// TwinCAT 3 PLC project automatedAquariumfilter
// ProgramVersion: 3.1.4024.0
// libraries:
//   Tc2_Standard, * (Beckhoff Automation GmbH)
//   Tc2_System, * (Beckhoff Automation GmbH)
//   Tc3_Module, * (Beckhoff Automation GmbH)
//   VisuDialogs, * (System)
//   VisuSymbols,3.5.10.0,System
// project tree:
//   FUNCTIONSBLOCKS/ FB_CO2.TcPOU, FB_FILTER.TcPOU, FB_HEATING.TcPOU, FB_LIGHT.TcPOU, FB_WATERCOOLING.TcPOU
//   / GlobalTextList.TcGTLO, GVL.TcGVL, PlcTask.TcTTO, Task_heat.TcTTO, Task_temp_monitor.TcTTO, Visualization Manager.TcVMO (not stored)
//   POUs/ HEATING.TcPOU, MAIN.TcPOU, TEMP_MONITOR.TcPOU
//   VISUs/ Visualization.TcVIS
// real-time tasks:
//   TASK PlcTask: cycle T#10ms, priority 20, ADS port 350

CONFIGURATION automatedAquariumfilter
    RESOURCE PLC ON TwinCAT3
        TASK PlcTask(INTERVAL := T#10ms, PRIORITY := 1);
        TASK Task_heat(INTERVAL := T#10ms, PRIORITY := 3);
        TASK Task_temp_monitor(INTERVAL := T#10ms, PRIORITY := 2);
        PROGRAM MAIN WITH PlcTask : MAIN;
        PROGRAM HEATING WITH Task_heat : HEATING;
        PROGRAM TEMP_MONITOR WITH Task_temp_monitor : TEMP_MONITOR;
    END_RESOURCE
END_CONFIGURATION

// ---- GVL.TcGVL
{attribute 'qualified_only'}
VAR_GLOBAL
	ix_START :BOOL;
	
	ox_FILTER_WATER: BOOL;
	ox_HEATER: BOOL;
	id_TEMP_SENSOR: DINT:=20;
	ix_COOLDOWN: BOOL;
	ix_TEMPRESET: BOOL;
	
	ox_CO2: BOOL;
	ox_LIGHT: BOOL;
	id_TEMP_SETPOINT: DINT:=28;
END_VAR

// ---- POUs/MAIN.TcPOU
PROGRAM MAIN
VAR
	FilterCycle1 : FB_FILTER;  // instantie van FB

	CO2_1:FB_CO2;
	LIGHT1:FB_LIGHT;
	
	
END_VAR

GVL.id_TEMP_SETPOINT:=28;

IF GVL.ix_TEMPRESET THEN
	GVL.id_TEMP_SENSOR := 30;
	GVL.ix_TEMPRESET:=FALSE;
END_IF

IF GVL.ix_COOLDOWN THEN
	GVL.id_TEMP_SENSOR := GVL.id_TEMP_SENSOR -5;
	GVL.ix_COOLDOWN:=FALSE;
END_IF	

GVL.ox_CO2 :=CO2_1.CO2;
GVL.ox_FILTER_WATER := FilterCycle1.FILTER_WATER;
GVL.ox_LIGHT :=LIGHT1.LIGHT;

//FUNCTIEBLOKKEN

FilterCycle1(ix_START := GVL.ix_START);
CO2_1(ix_START :=GVL.ix_START);
LIGHT1(ix_START :=GVL.ix_START);

END_PROGRAM

// ---- FUNCTIONSBLOCKS/FB_FILTER.TcPOU
FUNCTION_BLOCK FB_FILTER
VAR_INPUT
    ix_START : BOOL;  // HMI start input

END_VAR
VAR_OUTPUT
    FILTER_WATER : BOOL;  // output naar MAIN/HMI
END_VAR
VAR
    STATE_FILTER : INT := 0;  // interne state
    T_CYCLE : TON; 
    elapsed_ms : UDINT;  // elapsed time in ms
    cycle_ms   : UDINT;  // 5-second repeating cycle
END_VAR

// --- CASE state machine ---
CASE STATE_FILTER OF

    0: // Idle
        FILTER_WATER := FALSE;

        // Stop cycle timer
        T_CYCLE(IN := FALSE);

        // Start cycle
        IF ix_START THEN
            STATE_FILTER := 1;
        END_IF;

    1: // 30s cycle running
        // Abort cycle if button released
        IF ix_START = FALSE THEN
            STATE_FILTER := 0;
        END_IF;

        // Start 30-second timer
        T_CYCLE(IN := TRUE, PT := T#30S);
	
		// Convert elapsed time to milliseconds
		elapsed_ms := TO_UDINT(T_CYCLE.ET);

		// Create repeating 5-second cycle
		cycle_ms := elapsed_ms MOD 5000; // 5000 ms = 5 seconds
		
		// 0-3s -> ON, 3-5s -> OFF
		IF cycle_ms < 3000 THEN
			FILTER_WATER := TRUE;
		ELSE
			FILTER_WATER := FALSE;
		END_IF;
		        // End of cycle
        IF T_CYCLE.Q THEN
            STATE_FILTER := 0;
        END_IF;
       
END_CASE;

END_FUNCTION_BLOCK

// ---- FUNCTIONSBLOCKS/FB_CO2.TcPOU
FUNCTION_BLOCK FB_CO2
VAR_INPUT
	ix_START: BOOL;
END_VAR
VAR_OUTPUT
	CO2: BOOL;
END_VAR
VAR
	STATE: INT;
	T_CYCLE: TON;
END_VAR

// --- CASE state machine ---
CASE STATE OF

    0: // Idle
        CO2 := FALSE;
        // Stop cycle timer
        T_CYCLE(IN := FALSE);
        // Start cycle
        IF ix_START THEN
            STATE := 1;
        END_IF;
    1: // Start 30s cycle
        // Stop cycle if start button released
        IF ix_START = FALSE THEN
            STATE := 0;
        END_IF;
        // Start timer
        T_CYCLE(IN := TRUE, PT := T#30S);
        // Timed outputs
        CO2 := TRUE;
        // CO2 timing: ON at 10s, OFF at 20s
        IF (T_CYCLE.ET >= T#5S) AND (T_CYCLE.ET < T#20S) THEN
            CO2 := TRUE;
        ELSE
            CO2 := FALSE;
        END_IF;
        // End of cycle
        IF T_CYCLE.Q THEN
            STATE := 0;
        END_IF;
END_CASE;

END_FUNCTION_BLOCK

// ---- FUNCTIONSBLOCKS/FB_LIGHT.TcPOU
FUNCTION_BLOCK FB_LIGHT
VAR_INPUT

	ix_START: BOOL;
END_VAR
VAR_OUTPUT
	LIGHT: BOOL;
END_VAR
VAR
	STATE: INT;
	T_CYCLE: TON;
END_VAR

// --- CASE state machine ---
CASE STATE OF
    0: // Idle
        LIGHT := FALSE;
        // Stop cycle timer
        T_CYCLE(IN := FALSE);
        // Start cycle
        IF ix_START THEN
            STATE := 1;
        END_IF;
    1: // Start 30s cycle
        // Stop cycle if start button released
        IF ix_START = FALSE THEN
            STATE := 0;
        END_IF;
        // Start timer
        T_CYCLE(IN := TRUE, PT := T#30S);
        // Timed outputs
        LIGHT := TRUE;
        // LIGHT timing: ON at 10s, OFF at 25s
        IF (T_CYCLE.ET >= T#10S) AND (T_CYCLE.ET < T#25S) THEN
            LIGHT := TRUE;
        ELSE
            LIGHT := FALSE;
        END_IF;
        // End of cycle
        IF T_CYCLE.Q THEN
            STATE := 0;
        END_IF;
END_CASE;

END_FUNCTION_BLOCK

// ---- POUs/HEATING.TcPOU
PROGRAM HEATING
VAR
	HEATING1:FB_HEATING;
END_VAR


// GVL output koppelen
GVL.ox_HEATER :=HEATING1.HEATING;

HEATING1(ix_START:=GVL.ix_START,TEMP:=GVL.id_TEMP_SENSOR,
SETPOINT:=GVL.id_TEMP_SETPOINT);

END_PROGRAM

// ---- FUNCTIONSBLOCKS/FB_HEATING.TcPOU
FUNCTION_BLOCK FB_HEATING
VAR_INPUT
	ix_START: BOOL;
	TEMP: DINT;
	SETPOINT: DINT;
END_VAR
VAR_OUTPUT
	HEATING:BOOL;
END_VAR
VAR
	STATE: INT;
END_VAR

CASE STATE OF
	0: // Idle
        HEATING := FALSE;
        // Start cycle
        IF ix_START THEN
            STATE := 1;
        END_IF;
    1:
        IF ix_START = FALSE THEN
            STATE := 0;
        END_IF;
        IF (TEMP < SETPOINT) THEN
			HEATING :=TRUE;
		ELSE
			HEATING :=FALSE;
		END_IF
END_CASE;

END_FUNCTION_BLOCK

// ---- POUs/TEMP_MONITOR.TcPOU
PROGRAM TEMP_MONITOR
VAR
		WaterCooling1: FB_WATERCOOLING;	
END_VAR

WaterCooling1(HEATER:=GVL.ox_HEATER,TEMP_SENSOR:=GVL.id_TEMP_SENSOR);

END_PROGRAM

// ---- FUNCTIONSBLOCKS/FB_WATERCOOLING.TcPOU
FUNCTION_BLOCK FB_WATERCOOLING
VAR_INPUT
    HEATER : BOOL;          // Verwarming aan/uit
END_VAR

VAR_IN_OUT
    TEMP_SENSOR : DINT;      // Sensorwaarde in GVL
END_VAR

VAR
    T_TEMP : TON;           // 2-second timer
END_VAR


// --- Timer starten ---
T_TEMP(IN := TRUE, PT := T#2S);

// --- Temperature simulation ---
IF T_TEMP.Q THEN
    
    // Heating or cooling
    IF HEATER THEN
        TEMP_SENSOR := TEMP_SENSOR + 1;       // heat up
    ELSIF TEMP_SENSOR > 15 THEN
        TEMP_SENSOR := TEMP_SENSOR - 1;       // cool down
    END_IF;

    // Reset timer
    T_TEMP(IN := FALSE);
END_IF;

END_FUNCTION_BLOCK

// ---- GlobalTextList.TcGTLO
TEXTLIST GlobalTextList
  414 = 'AAN/UIT'
  444 = 'CO2'
  71 = 'FILTER CO2'
  565 = 'FILTER WATER'
  363 = 'HEATER'
  99 = 'LIGHT'
  961 = 'SETPOINT T: %d °C'
  157 = 'START'
  656 = 'Temperature: %d °C'
  219 = 'Temperature: %I °C'
  935 = 'Temperature: %I0 °C'
  355 = 'TIME: %d sec'
  206 = 'TIME: %t sec'
  667 = 'TIME: %t[m:s:ms]'
  721 = 'TIME: %t[m:s:ms}'
  125 = 'TIME: %t[m:s:ms}m:s:ms '
  648 = 'TIME: %t[m:s]'
  562 = 'TIME: %t[s:ms]'
  683 = 'WATER T%d °C'
  33 = 'WATER T: %d °C'
  372 = 'water temperature -5'
  29 = 'water temperature -5°C'
  245 = 'water temperature 30°C'
END_TEXTLIST

// ---- VISUs/Visualization.TcVIS
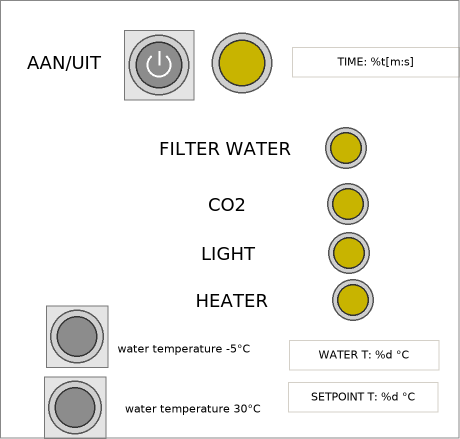
VISUALIZATION Visualization  // 460x439
    Lamp1 (207,28 70x70), variable: GVL.ix_START, style: Lamp-Lamp1-Yellow
    PowerSwitch (124,30 70x70), variable: GVL.ix_START, behaviour: TOGGLE, style: Switch-PowerSwitch-Gray
    Label (14,48 101x30), "AAN/UIT"
    Lamp1 (322,124 48x48), variable: GVL.ox_FILTER_WATER, style: Lamp-Lamp1-Yellow
    Textfield (288,382 150x30), "SETPOINT T: %d °C", text variable: GVL.id_TEMP_SETPOINT
    PushSwitch (46,305 62x63), variable: GVL.ix_COOLDOWN, behaviour: TOGGLE, style: Switch-PushSwitch-Gray
    Label (109,334 150x30), "water temperature -5°C"
    Label (138,134 174x30), "FILTER WATER"
    Lamp1 (324,180 48x48), variable: GVL.ox_CO2, style: Lamp-Lamp1-Yellow
    Label (140,190 174x30), "CO2"
    Lamp1 (325,229 48x48), variable: GVL.ox_LIGHT, style: Lamp-Lamp1-Yellow
    Label (141,239 174x30), "LIGHT"
    Lamp1 (329,276 48x48), variable: GVL.ox_HEATER, style: Lamp-Lamp1-Yellow
    Label (145,286 174x30), "HEATER"
    PushSwitch (44,376 62x63), variable: GVL.ix_TEMPRESET, behaviour: TOGGLE, style: Switch-PushSwitch-Gray
    Label (118,394 150x30), "water temperature 30°C"
    Textfield (292,47 168x30), "TIME: %t[m:s]", text variable: MAIN.FilterCycle1.T_CYCLE.ET
    Textfield (289,340 150x30), "WATER T: %d °C", text variable: GVL.id_TEMP_SENSOR
END_VISUALIZATION
